TYPE E_EndoscopePosture:
(
	EndoscopePosture_HeadUp:=1,
	EndoScopePosture_HeadDown:=2
);
END_TYPE

(* stored: Version 1.1.0.1, ProductVersion 3.1.4024.11
   DUT E_EndoscopePosture: Id {deeaab70-706a-4203-af52-30ab29d02ff5} *)
